PROGRAM MAIN
VAR
	//cmt1
	bTest: BOOL;
END_VAR

END_PROGRAM

(* stored: Version 1.1.0.1, ProductVersion 3.1.4024.11
   POU MAIN: Id {30f9bb9c-f662-48d2-897d-ecb9b184900d}, SpecialFunc None *)
